Staubli VAL3: lists.pjx

--- lists.pjx ---
Parameters version=s8.13.1Cs9_BS2800 stackSize=5000 millimeterUnit=true
Data file=lists.dtx

--- lists.dtx ---
mdesc mNomSpeed
public string sString
